// TIA Portal V21 export
TYPE "LBC_typeMotorStarterProcessValues"
TITLE = LBC_typeMotorStarterProcessValues
// Module related monitoring information
   STRUCT
      enable { ExternalWritable := 'False'} : Bool;   // Enable functionality of FB
      referenceDesignator { ExternalWritable := 'False'} : WString[154];   // Reference Designator for the module incl. its parent
      enabledStarter { ExternalWritable := 'False'} : Bool;   // Start/enable the motor starter
      resetStarter { ExternalWritable := 'False'} : Bool;   // Reset the starter in case of an active `error` and command `resetStarter`
      starterActive { ExternalWritable := 'False'} : Bool;   // Starter is switched on and `feedbackReady`is present
      commandForward { ExternalWritable := 'False'} : Bool;   // Start the motor forward
      commandBackward { ExternalWritable := 'False'} : Bool;   // Start the motor backward
      reset { ExternalWritable := 'False'} : Bool;   // Command reset the motor starter
      forward { ExternalWritable := 'False'} : Bool;   // Starting the motor forward
      backward { ExternalWritable := 'False'} : Bool;   // Starting the motor backward
      feedbackReady { ExternalWritable := 'False'} : Bool;   // Motor is ready for switching on
      feedbackRunningForward { ExternalWritable := 'False'} : Bool;   // Motor is running / soft starter bypass in forward direction
      feedbackRunningBackward { ExternalWritable := 'False'} : Bool;   // Motor is running / soft starter bypass in backward direction
      feedbackError { ExternalWritable := 'False'} : Bool;   // Motor starter is in error state (e.g. overheating)
      interlock { ExternalWritable := 'False'} : Bool;   // TRUE: Normal operation, FALSE: Locking the operation mode
      interlockWarning { ExternalWritable := 'False'} : Bool;   // Prohibeted command requested denied during interlock
      valid { ExternalWritable := 'False'} : Bool;   // Valid set of output values available at the FB
      busy { ExternalWritable := 'False'} : Bool;   // FB is not finished and new output values can be expected
      error { ExternalWritable := 'False'} : Bool;   // An error occurred while processing the FB
      enableManualCmds { ExternalWritable := 'False'} : Bool;   // Enabling manual commands via interface
      status { ExternalWritable := 'False'} : Word;   // 16#0000-16#7FFF: Status of the FB 16#8000-16#FFFF: Error identification
   END_STRUCT;
END_TYPE
